(* IEC 61131-3 sources: sphere-usecases/water-treatment/implementations/openplc/projects/simulator_project, 4 files *)

(* ---- simulator_clean.st ---- *)
TYPE
  HMI_UDT : STRUCT
    Start_PB : BOOL;
    Stop_PB : BOOL;
    Start_Active : BOOL;
    Stop_Active : BOOL;
  END_STRUCT;
  P1_UDT : STRUCT
    RW_Tank_tnk_lvl : REAL;
    RW_Pump_flow : REAL;
    RW_Tank_PR_Valve_sts : BOOL;
    RW_Tank_P6B_Valve_sts : BOOL;
    RW_Tank_P_Valve_sts : BOOL;
    RW_Pump_sts : BOOL;
    RW_Pump_fault : BOOL;
    RW_Pump : REAL;
    RW_Tank_PR_Valve : BOOL;
    RW_Tank_P_Valve : BOOL;
    RW_Pump_start : BOOL;
    RW_Pump_stop : BOOL;
    RW_Tank_P6B_Valve : BOOL;
  END_STRUCT;
  P2_UDT : STRUCT
    ChemTreat_NaCl_Tank_tnk_lvl : REAL;
    ChemTreat_NaOCl_Tank_tnk_lvl : REAL;
    ChemTreat_HCl_Tank_tnk_lvl : REAL;
    ChemTreat_NaCl_Tank_Valve_sts : BOOL;
    ChemTreat_NaOCl_Tank_Valve_sts : BOOL;
    ChemTreat_HCl_Tank_Valve_sts : BOOL;
    ChemTreat_NaCl_Tank_Valve : BOOL;
    ChemTreat_NaOCl_Tank_Valve : BOOL;
    ChemTreat_HCl_Tank_Valve : BOOL;
  END_STRUCT;
  P3_UDT : STRUCT
    Ultrafiltration_UFFT_Tank_tnk_lvl : REAL;
    Ultrafiltration_UFFT_Tank_Valve_sts : BOOL;
    Ultrafiltration_UF_Drain_Valve_sts : BOOL;
    Ultrafiltration_UF_ROFT_Valve_sts : BOOL;
    Ultrafiltration_UF_BWP_Valve_sts : BOOL;
    Ultrafiltration_UFFT_Tank_Valve : BOOL;
    Ultrafiltration_UF_Drain_Valve : BOOL;
    Ultrafiltration_UF_ROFT_Valve : BOOL;
    Ultrafiltration_UF_BWP_Valve : BOOL;
  END_STRUCT;
  Phases_UDT : STRUCT
    Filling : BOOL;
    Draining : BOOL;
  END_STRUCT;
  RW_tank_AL_UDT : STRUCT
    LL_alarm : BOOL;
    L_alarm : BOOL;
    H_alarm : BOOL;
    HH_alarm : BOOL;
  END_STRUCT;
  System_State_UDT : STRUCT
    IDLE : BOOL;
    START : BOOL;
    RUNNING : BOOL;
    SHUTDOWN : BOOL;
    Permissives : ARRAY [0..31] OF BOOL;
    Permissives_Ready : BOOL;
  END_STRUCT;
  SYS_MESSAGES : STRUCT
    ProgramScanTime : DINT;
    AvailableMemory : REAL;
    ControllerStatus : SINT;
    ScanTime : REAL;
  END_STRUCT;
END_TYPE

PROGRAM MainProgram
  VAR_INPUT
    Alarms : RW_tank_AL_UDT;
    GSV_Message : SYS_MESSAGES;
    HMI : HMI_UDT;
    P1 : P1_UDT;
    P1_SYS : System_State_UDT;
    P2 : P2_UDT;
    P3 : P3_UDT;
  END_VAR
  VAR_INPUT
    di_2_0 AT %IX2.0 : BOOL;
    di_2_1 AT %IX2.1 : BOOL;
    di_2_10 AT %IX2.10 : BOOL;
    di_2_11 AT %IX2.11 : BOOL;
    di_2_2 AT %IX2.2 : BOOL;
    di_2_3 AT %IX2.3 : BOOL;
    di_2_4 AT %IX2.4 : BOOL;
    di_2_5 AT %IX2.5 : BOOL;
    di_2_6 AT %IX2.6 : BOOL;
    di_2_8 AT %IX2.8 : BOOL;
    di_2_9 AT %IX2.9 : BOOL;
    ai_7_0 AT %IW70 : REAL;
    di_7_ch0halarm AT %IX7.0 : BOOL;
    di_7_ch0hhalarm AT %IX7.0 : BOOL;
    di_7_ch0lalarm AT %IX7.0 : BOOL;
    di_7_ch0llalarm AT %IX7.0 : BOOL;
    ai_7_1 AT %IW71 : REAL;
    ai_7_2 AT %IW72 : REAL;
    ai_7_3 AT %IW73 : REAL;
    ai_7_4 AT %IW74 : REAL;
    ai_7_5 AT %IW75 : REAL;
  END_VAR
  VAR_OUTPUT
    ao_10_0 AT %QW100 : REAL;
    do_5_0 AT %QX5.0 : BOOL;
    do_5_1 AT %QX5.1 : BOOL;
    do_5_10 AT %QX5.10 : BOOL;
    do_5_11 AT %QX5.11 : BOOL;
    do_5_2 AT %QX5.2 : BOOL;
    do_5_3 AT %QX5.3 : BOOL;
    do_5_4 AT %QX5.4 : BOOL;
    do_5_5 AT %QX5.5 : BOOL;
    do_5_6 AT %QX5.6 : BOOL;
    do_5_7 AT %QX5.7 : BOOL;
    do_5_8 AT %QX5.8 : BOOL;
    do_5_9 AT %QX5.9 : BOOL;
  END_VAR

  (* IO_setup *)
  (* P1 Analog Input *)
  P1.RW_Tank_tnk_lvl := ai_7_0;
  P1.RW_Pump_flow := ai_7_1;
  (* P1 Digital Input *)
  P1.RW_Tank_PR_Valve_sts := di_2_0;
  P1.RW_Tank_P6B_Valve_sts := di_2_1;
  P1.RW_Tank_P_Valve_sts := di_2_2;
  P1.RW_Pump_sts := di_2_3;
  P1.RW_Pump_fault := di_2_4;
  (* P1 Analog Output *)
  P1.RW_Pump := ao_10_0;
  (* Digital Output *)
  P1.RW_Tank_PR_Valve := do_5_0;
  P1.RW_Tank_P6B_Valve := do_5_1;
  P1.RW_Tank_P_Valve := do_5_2;
  P1.RW_Pump_start := do_5_3;
  P1.RW_Pump_stop := do_5_4;
  (* P1 raw water tank alarms *)
  Alarms.LL_alarm := di_7_ch0llalarm;
  Alarms.L_alarm := di_7_ch0lalarm;
  Alarms.H_alarm := di_7_ch0halarm;
  Alarms.HH_alarm := di_7_ch0hhalarm;
  (* P2 Analog Input *)
  P2.ChemTreat_NaCl_Tank_tnk_lvl := ai_7_2;
  P2.ChemTreat_NaOCl_Tank_tnk_lvl := ai_7_3;
  P2.ChemTreat_HCl_Tank_tnk_lvl := ai_7_4;
  (* P2 Digital Input *)
  P2.ChemTreat_NaCl_Tank_Valve_sts := di_2_5;
  P2.ChemTreat_NaOCl_Tank_Valve_sts := di_2_6;
  (* P2 Analog Output *)
  (* NONE *)
  (* P2 Digital Output *)
  P2.ChemTreat_NaCl_Tank_Valve := do_5_5;
  P2.ChemTreat_NaOCl_Tank_Valve := do_5_6;
  P2.ChemTreat_HCl_Tank_Valve := do_5_7;
  (* P3 Analog Input *)
  P3.Ultrafiltration_UFFT_Tank_tnk_lvl := ai_7_5;
  (* P3 Digital Input *)
  P3.Ultrafiltration_UFFT_Tank_Valve_sts := di_2_8;
  P3.Ultrafiltration_UF_Drain_Valve_sts := di_2_9;
  P3.Ultrafiltration_UF_Drain_Valve_sts := di_2_10;
  P3.Ultrafiltration_UF_BWP_Valve_sts := di_2_11;
  (* P3 Analog Output *)
  (* none *)
  (* P3 Digital Output *)
  P3.Ultrafiltration_UFFT_Tank_Valve := do_5_8;
  P3.Ultrafiltration_UF_Drain_Valve := do_5_9;
  P3.Ultrafiltration_UF_ROFT_Valve := do_5_10;
  P3.Ultrafiltration_UF_BWP_Valve := do_5_11;

  (* Raw_water_control *)
  if P1.RW_Tank_tnk_lvl = 250.0 and P1_SYS.RUNNING then
  P1.RW_Pump_stop := True;
  P1.RW_Pump_start := False; (* send the outputs *)
  Alarms.LL_alarm := True;
  (* if the level is at 500 or lower than 500 open the valve *)
  elsif P1.RW_Tank_tnk_lvl <= 500.0 and P1_SYS.RUNNING then
  (* output to turn the valve open *)
  P1.RW_Tank_PR_Valve := True;
  Alarms.L_alarm := True;
  (* if level is at 800 *)
  elsif  P1.RW_Tank_tnk_lvl = 800.0 and P1_SYS.RUNNING then
  P1.RW_Tank_PR_Valve := False; (* close the valve *)
  Alarms.H_alarm := True;
  elsif P1.RW_Tank_tnk_lvl = 1200.0 and P1_SYS.RUNNING then
  Alarms.HH_alarm := True; (* if the tank is higher than or equal to 1200 set the high high alarm *)
  end_if;

  (* Raw_water_pump *)
  if P3.Ultrafiltration_UFFT_Tank_tnk_lvl = 800.0 AND P1_SYS.RUNNING then
  (* start the pump and open the valve from the other tank *)
  P1.RW_Tank_P_Valve := True;
  P1.RW_Pump_start := True;
  P1.RW_Pump_stop := False;
  elsif P3.Ultrafiltration_UFFT_Tank_tnk_lvl = 1000.0 AND P1_SYS.RUNNING then
  (* stop the pump and close the valve *)
  P1.RW_Tank_P_Valve := False;
  P1.RW_Pump_stop := True;
  P1.RW_Pump_start := False;
  end_if;

  (* State_change *)
  if not HMI.Start_Active AND not HMI.Stop_Active then
  (* if start and stop is not pressed go to idle *)
  P1_SYS.IDLE := True;
  P1_SYS.START := False;
  P1_SYS.RUNNING := False;
  P1_SYS.SHUTDOWN := False;
  elsif  HMI.Start_Active AND not HMI.Stop_Active then
  (* if the start pb and stop is not pressed then change the state of process one to starting *)
  P1_SYS.IDLE := False;
  P1_SYS.START := True;
  P1_SYS.RUNNING := False;
  P1_SYS.SHUTDOWN := False;
  (* if the tank level is greater than 250 at the start and UFFT is less than a 1000 we can start *)
  (* then and all permissves cond together into one tag so we know the plant is ready to start *)
  P1_SYS.Permissives_Ready := P1_SYS.Permissives[0] AND P1_SYS.Permissives[1];
  elsif HMI.Start_Active AND P1_SYS.Permissives_Ready then
  (* if the start was pressed and permissives are ready start running Process one *)
  P1_SYS.IDLE := False;
  P1_SYS.START := False;
  P1_SYS.RUNNING := True;
  P1_SYS.SHUTDOWN := False;
  elsif HMI.Stop_Active then
  (* if the stop button is pressed then go to shutdown state *)
  P1_SYS.IDLE := False;
  P1_SYS.START := False;
  P1_SYS.RUNNING := False;
  P1_SYS.SHUTDOWN := True;
  (* set all permissives to false *)
  P1_SYS.Permissives_Ready := False;
  end_if;
END_PROGRAM

CONFIGURATION config
  VAR_GLOBAL
    ao_10_0 AT %QW100 : REAL;
    di_2_0 AT %IX2.0 : BOOL;
    di_2_1 AT %IX2.1 : BOOL;
    di_2_10 AT %IX2.10 : BOOL;
    di_2_11 AT %IX2.11 : BOOL;
    di_2_2 AT %IX2.2 : BOOL;
    di_2_3 AT %IX2.3 : BOOL;
    di_2_4 AT %IX2.4 : BOOL;
    di_2_5 AT %IX2.5 : BOOL;
    di_2_6 AT %IX2.6 : BOOL;
    di_2_8 AT %IX2.8 : BOOL;
    di_2_9 AT %IX2.9 : BOOL;
    do_5_0 AT %QX5.0 : BOOL;
    do_5_1 AT %QX5.1 : BOOL;
    do_5_10 AT %QX5.10 : BOOL;
    do_5_11 AT %QX5.11 : BOOL;
    do_5_2 AT %QX5.2 : BOOL;
    do_5_3 AT %QX5.3 : BOOL;
    do_5_4 AT %QX5.4 : BOOL;
    do_5_5 AT %QX5.5 : BOOL;
    do_5_6 AT %QX5.6 : BOOL;
    do_5_7 AT %QX5.7 : BOOL;
    do_5_8 AT %QX5.8 : BOOL;
    do_5_9 AT %QX5.9 : BOOL;
    ai_7_0 AT %IW70 : REAL;
    di_7_ch0halarm AT %IX7.0 : BOOL;
    di_7_ch0hhalarm AT %IX7.0 : BOOL;
    di_7_ch0lalarm AT %IX7.0 : BOOL;
    di_7_ch0llalarm AT %IX7.0 : BOOL;
    ai_7_1 AT %IW71 : REAL;
    ai_7_2 AT %IW72 : REAL;
    ai_7_3 AT %IW73 : REAL;
    ai_7_4 AT %IW74 : REAL;
    ai_7_5 AT %IW75 : REAL;
  END_VAR

  RESOURCE res_MainProgram ON PLC
    TASK task_MainProgram(INTERVAL := T#100ms,PRIORITY := 0);
    PROGRAM MainProgram_instance : MainProgram;
  END_RESOURCE
END_CONFIGURATION

(* ---- simulator_final.st ---- *)
PROGRAM SimulatorProgram
  VAR
    (* ===== Internal physics state ===== *)
    rw_tank_level : REAL := 600.0;
    uf_tank_level : REAL := 400.0;
    nacl_level : REAL := 800.0;
    naocl_level : REAL := 800.0;
    hcl_level : REAL := 800.0;
    pump_running : BOOL := FALSE;
    pump_flow : REAL := 0.0;

    (* Valve status with delay timers *)
    pr_valve_open : BOOL := FALSE;
    pr_valve_timer : INT := 0;
    p6b_valve_open : BOOL := FALSE;
    p6b_valve_timer : INT := 0;
    p_valve_open : BOOL := FALSE;
    p_valve_timer : INT := 0;
    nacl_valve_open : BOOL := FALSE;
    nacl_valve_timer : INT := 0;
    naocl_valve_open : BOOL := FALSE;
    naocl_valve_timer : INT := 0;
    hcl_valve_open : BOOL := FALSE;
    hcl_valve_timer : INT := 0;
    uf_valve_open : BOOL := FALSE;
    uf_valve_timer : INT := 0;
    uf_drain_open : BOOL := FALSE;
    uf_drain_timer : INT := 0;
    uf_roft_open : BOOL := FALSE;
    uf_roft_timer : INT := 0;
    uf_bwp_open : BOOL := FALSE;
    uf_bwp_timer : INT := 0;

    init_done : BOOL := FALSE;
    pump_timer : INT := 0;
    pump_requested : BOOL := FALSE;
    admin_reset_seq_seen : INT := 0;
    admin_apply_seq_seen : INT := 0;

    (* ===== Constants ===== *)
    DT_SEC : REAL := 0.1;            (* 100ms scan interval *)
    PUMP_MAX_FLOW : REAL := 120.0;   (* L/min at 100% speed *)
    PR_INFLOW_RATE : REAL := 50.0;   (* L/min from external source *)
    DOSING_RATE : REAL := 5.0;       (* L/min chemical drain *)
    UF_DRAIN_RATE : REAL := 30.0;    (* L/min UF drain/ROFT *)
    VALVE_DELAY : INT := 5;          (* cycles = 500ms *)
    PUMP_DELAY : INT := 8;           (* cycles = 800ms *)
    RW_TANK_MAX : REAL := 1500.0;
    UF_TANK_MAX : REAL := 1200.0;
    CHEM_TANK_MAX : REAL := 1000.0;
  END_VAR
  VAR_EXTERNAL
    (* ===== Bridge command inputs - written by external bridge ===== *)
    cmd_pr_valve : INT;      (* 0/1  PR valve command *)
    cmd_p6b_valve : INT;     (* 0/1  P6B valve command *)
    cmd_p_valve : INT;       (* 0/1  Process valve command *)
    cmd_pump_start : INT;    (* 0/1  Pump start *)
    cmd_pump_stop : INT;     (* 0/1  Pump stop *)
    cmd_nacl_valve : INT;    (* 0/1  NaCl valve command *)
    cmd_naocl_valve : INT;   (* 0/1  NaOCl valve command *)
    cmd_hcl_valve : INT;     (* 0/1  HCl valve command *)
    cmd_uf_valve : INT;      (* 0/1  UF tank valve command *)
    cmd_uf_drain : INT;      (* 0/1  UF drain valve command *)
    cmd_uf_roft : INT;       (* 0/1  UF ROFT valve command *)
    cmd_uf_bwp : INT;        (* 0/1  UF BWP valve command *)
    cmd_pump_speed : INT;    (* 0-100  pump speed % *)
    admin_init_rw_level : INT;   (* reset baseline: RW tank level *)
    admin_init_uf_level : INT;   (* reset baseline: UF tank level *)
    admin_init_nacl_level : INT; (* reset baseline: NaCl tank *)
    admin_init_naocl_level : INT;(* reset baseline: NaOCl tank *)
    admin_init_hcl_level : INT;  (* reset baseline: HCl tank *)
    admin_reset_seq : INT;       (* increments trigger full sim reset *)
    admin_apply_rw_level : INT;  (* runtime RW level override *)
    admin_apply_uf_level : INT;  (* runtime UF level override *)
    admin_apply_nacl_level : INT;(* runtime NaCl level override *)
    admin_apply_naocl_level : INT;(* runtime NaOCl level override *)
    admin_apply_hcl_level : INT; (* runtime HCl level override *)
    admin_apply_rw_flag : INT;   (* 0/1 apply override *)
    admin_apply_uf_flag : INT;
    admin_apply_nacl_flag : INT;
    admin_apply_naocl_flag : INT;
    admin_apply_hcl_flag : INT;
    admin_apply_seq : INT;       (* increments trigger level apply *)

    (* ===== Bridge sensor outputs - read by bridge ===== *)
    out_rw_level : INT;      (* RW tank level mm *)
    out_rw_flow : INT;       (* RW pump flow L/min *)
    out_nacl_level : INT;    (* NaCl tank level mm *)
    out_naocl_level : INT;   (* NaOCl tank level mm *)
    out_hcl_level : INT;     (* HCl tank level mm *)
    out_uf_level : INT;      (* UF tank level mm *)
    out_pr_valve_sts : INT;  (* 0/1 *)
    out_p6b_valve_sts : INT;
    out_p_valve_sts : INT;
    out_pump_sts : INT;
    out_pump_fault : INT;
    out_nacl_valve_sts : INT;
    out_naocl_valve_sts : INT;
    out_hcl_valve_sts : INT;
    out_uf_valve_sts : INT;
    out_uf_drain_sts : INT;
    out_uf_roft_sts : INT;
    out_uf_bwp_sts : INT;
  END_VAR

  IF NOT init_done THEN
    rw_tank_level := 600.0;
    uf_tank_level := 400.0;
    nacl_level := 800.0;
    naocl_level := 800.0;
    hcl_level := 800.0;
    pump_running := FALSE;
    pump_flow := 0.0;
    pr_valve_open := FALSE;
    pr_valve_timer := 0;
    p6b_valve_open := FALSE;
    p6b_valve_timer := 0;
    p_valve_open := FALSE;
    p_valve_timer := 0;
    nacl_valve_open := FALSE;
    nacl_valve_timer := 0;
    naocl_valve_open := FALSE;
    naocl_valve_timer := 0;
    hcl_valve_open := FALSE;
    hcl_valve_timer := 0;
    uf_valve_open := FALSE;
    uf_valve_timer := 0;
    uf_drain_open := FALSE;
    uf_drain_timer := 0;
    uf_roft_open := FALSE;
    uf_roft_timer := 0;
    uf_bwp_open := FALSE;
    uf_bwp_timer := 0;
    pump_timer := 0;
    pump_requested := FALSE;
    admin_reset_seq_seen := admin_reset_seq;
    admin_apply_seq_seen := admin_apply_seq;
    init_done := TRUE;
  END_IF;

  (* ========================================================= *)
  (* 0. Testbed admin hooks                                    *)
  (*    These registers let the host reset or perturb the sim  *)
  (*    without rebuilding images or restarting the stack.     *)
  (* ========================================================= *)
  IF admin_reset_seq <> admin_reset_seq_seen THEN
    admin_reset_seq_seen := admin_reset_seq;
    rw_tank_level := INT_TO_REAL(admin_init_rw_level);
    uf_tank_level := INT_TO_REAL(admin_init_uf_level);
    nacl_level := INT_TO_REAL(admin_init_nacl_level);
    naocl_level := INT_TO_REAL(admin_init_naocl_level);
    hcl_level := INT_TO_REAL(admin_init_hcl_level);
    pump_running := FALSE;
    pump_flow := 0.0;
    pr_valve_open := FALSE;
    pr_valve_timer := 0;
    p6b_valve_open := FALSE;
    p6b_valve_timer := 0;
    p_valve_open := FALSE;
    p_valve_timer := 0;
    nacl_valve_open := FALSE;
    nacl_valve_timer := 0;
    naocl_valve_open := FALSE;
    naocl_valve_timer := 0;
    hcl_valve_open := FALSE;
    hcl_valve_timer := 0;
    uf_valve_open := FALSE;
    uf_valve_timer := 0;
    uf_drain_open := FALSE;
    uf_drain_timer := 0;
    uf_roft_open := FALSE;
    uf_roft_timer := 0;
    uf_bwp_open := FALSE;
    uf_bwp_timer := 0;
    pump_timer := 0;
    pump_requested := FALSE;
  END_IF;

  IF admin_apply_seq <> admin_apply_seq_seen THEN
    admin_apply_seq_seen := admin_apply_seq;
    IF admin_apply_rw_flag <> 0 THEN
      rw_tank_level := INT_TO_REAL(admin_apply_rw_level);
    END_IF;
    IF admin_apply_uf_flag <> 0 THEN
      uf_tank_level := INT_TO_REAL(admin_apply_uf_level);
    END_IF;
    IF admin_apply_nacl_flag <> 0 THEN
      nacl_level := INT_TO_REAL(admin_apply_nacl_level);
    END_IF;
    IF admin_apply_naocl_flag <> 0 THEN
      naocl_level := INT_TO_REAL(admin_apply_naocl_level);
    END_IF;
    IF admin_apply_hcl_flag <> 0 THEN
      hcl_level := INT_TO_REAL(admin_apply_hcl_level);
    END_IF;
  END_IF;

  (* ========================================================= *)
  (* 1. Update valve status with delay                         *)
  (* ========================================================= *)

  (* PR valve *)
  IF cmd_pr_valve <> 0 THEN
    IF NOT pr_valve_open THEN
      pr_valve_timer := pr_valve_timer + 1;
      IF pr_valve_timer >= VALVE_DELAY THEN
        pr_valve_open := TRUE;
        pr_valve_timer := 0;
      END_IF;
    END_IF;
  ELSE
    IF pr_valve_open THEN
      pr_valve_timer := pr_valve_timer + 1;
      IF pr_valve_timer >= VALVE_DELAY THEN
        pr_valve_open := FALSE;
        pr_valve_timer := 0;
      END_IF;
    ELSE
      pr_valve_timer := 0;
    END_IF;
  END_IF;

  (* P6B valve *)
  IF cmd_p6b_valve <> 0 THEN
    IF NOT p6b_valve_open THEN
      p6b_valve_timer := p6b_valve_timer + 1;
      IF p6b_valve_timer >= VALVE_DELAY THEN
        p6b_valve_open := TRUE;
        p6b_valve_timer := 0;
      END_IF;
    END_IF;
  ELSE
    IF p6b_valve_open THEN
      p6b_valve_timer := p6b_valve_timer + 1;
      IF p6b_valve_timer >= VALVE_DELAY THEN
        p6b_valve_open := FALSE;
        p6b_valve_timer := 0;
      END_IF;
    ELSE
      p6b_valve_timer := 0;
    END_IF;
  END_IF;

  (* P valve *)
  IF cmd_p_valve <> 0 THEN
    IF NOT p_valve_open THEN
      p_valve_timer := p_valve_timer + 1;
      IF p_valve_timer >= VALVE_DELAY THEN
        p_valve_open := TRUE;
        p_valve_timer := 0;
      END_IF;
    END_IF;
  ELSE
    IF p_valve_open THEN
      p_valve_timer := p_valve_timer + 1;
      IF p_valve_timer >= VALVE_DELAY THEN
        p_valve_open := FALSE;
        p_valve_timer := 0;
      END_IF;
    ELSE
      p_valve_timer := 0;
    END_IF;
  END_IF;

  (* NaCl valve *)
  IF cmd_nacl_valve <> 0 THEN
    IF NOT nacl_valve_open THEN
      nacl_valve_timer := nacl_valve_timer + 1;
      IF nacl_valve_timer >= VALVE_DELAY THEN
        nacl_valve_open := TRUE;
        nacl_valve_timer := 0;
      END_IF;
    END_IF;
  ELSE
    IF nacl_valve_open THEN
      nacl_valve_timer := nacl_valve_timer + 1;
      IF nacl_valve_timer >= VALVE_DELAY THEN
        nacl_valve_open := FALSE;
        nacl_valve_timer := 0;
      END_IF;
    ELSE
      nacl_valve_timer := 0;
    END_IF;
  END_IF;

  (* NaOCl valve *)
  IF cmd_naocl_valve <> 0 THEN
    IF NOT naocl_valve_open THEN
      naocl_valve_timer := naocl_valve_timer + 1;
      IF naocl_valve_timer >= VALVE_DELAY THEN
        naocl_valve_open := TRUE;
        naocl_valve_timer := 0;
      END_IF;
    END_IF;
  ELSE
    IF naocl_valve_open THEN
      naocl_valve_timer := naocl_valve_timer + 1;
      IF naocl_valve_timer >= VALVE_DELAY THEN
        naocl_valve_open := FALSE;
        naocl_valve_timer := 0;
      END_IF;
    ELSE
      naocl_valve_timer := 0;
    END_IF;
  END_IF;

  (* HCl valve *)
  IF cmd_hcl_valve <> 0 THEN
    IF NOT hcl_valve_open THEN
      hcl_valve_timer := hcl_valve_timer + 1;
      IF hcl_valve_timer >= VALVE_DELAY THEN
        hcl_valve_open := TRUE;
        hcl_valve_timer := 0;
      END_IF;
    END_IF;
  ELSE
    IF hcl_valve_open THEN
      hcl_valve_timer := hcl_valve_timer + 1;
      IF hcl_valve_timer >= VALVE_DELAY THEN
        hcl_valve_open := FALSE;
        hcl_valve_timer := 0;
      END_IF;
    ELSE
      hcl_valve_timer := 0;
    END_IF;
  END_IF;

  (* UF tank valve *)
  IF cmd_uf_valve <> 0 THEN
    IF NOT uf_valve_open THEN
      uf_valve_timer := uf_valve_timer + 1;
      IF uf_valve_timer >= VALVE_DELAY THEN
        uf_valve_open := TRUE;
        uf_valve_timer := 0;
      END_IF;
    END_IF;
  ELSE
    IF uf_valve_open THEN
      uf_valve_timer := uf_valve_timer + 1;
      IF uf_valve_timer >= VALVE_DELAY THEN
        uf_valve_open := FALSE;
        uf_valve_timer := 0;
      END_IF;
    ELSE
      uf_valve_timer := 0;
    END_IF;
  END_IF;

  (* UF drain valve *)
  IF cmd_uf_drain <> 0 THEN
    IF NOT uf_drain_open THEN
      uf_drain_timer := uf_drain_timer + 1;
      IF uf_drain_timer >= VALVE_DELAY THEN
        uf_drain_open := TRUE;
        uf_drain_timer := 0;
      END_IF;
    END_IF;
  ELSE
    IF uf_drain_open THEN
      uf_drain_timer := uf_drain_timer + 1;
      IF uf_drain_timer >= VALVE_DELAY THEN
        uf_drain_open := FALSE;
        uf_drain_timer := 0;
      END_IF;
    ELSE
      uf_drain_timer := 0;
    END_IF;
  END_IF;

  (* UF ROFT valve *)
  IF cmd_uf_roft <> 0 THEN
    IF NOT uf_roft_open THEN
      uf_roft_timer := uf_roft_timer + 1;
      IF uf_roft_timer >= VALVE_DELAY THEN
        uf_roft_open := TRUE;
        uf_roft_timer := 0;
      END_IF;
    END_IF;
  ELSE
    IF uf_roft_open THEN
      uf_roft_timer := uf_roft_timer + 1;
      IF uf_roft_timer >= VALVE_DELAY THEN
        uf_roft_open := FALSE;
        uf_roft_timer := 0;
      END_IF;
    ELSE
      uf_roft_timer := 0;
    END_IF;
  END_IF;

  (* UF BWP valve *)
  IF cmd_uf_bwp <> 0 THEN
    IF NOT uf_bwp_open THEN
      uf_bwp_timer := uf_bwp_timer + 1;
      IF uf_bwp_timer >= VALVE_DELAY THEN
        uf_bwp_open := TRUE;
        uf_bwp_timer := 0;
      END_IF;
    END_IF;
  ELSE
    IF uf_bwp_open THEN
      uf_bwp_timer := uf_bwp_timer + 1;
      IF uf_bwp_timer >= VALVE_DELAY THEN
        uf_bwp_open := FALSE;
        uf_bwp_timer := 0;
      END_IF;
    ELSE
      uf_bwp_timer := 0;
    END_IF;
  END_IF;

  (* ========================================================= *)
  (* 2. Update pump status with delay                          *)
  (* ========================================================= *)
  pump_requested := cmd_pump_start <> 0 AND cmd_pump_stop = 0;

  IF pump_requested AND NOT pump_running THEN
    pump_timer := pump_timer + 1;
    IF pump_timer >= PUMP_DELAY THEN
      pump_running := TRUE;
      pump_timer := 0;
    END_IF;
  ELSIF NOT pump_requested AND pump_running THEN
    pump_timer := pump_timer + 1;
    IF pump_timer >= PUMP_DELAY THEN
      pump_running := FALSE;
      pump_timer := 0;
    END_IF;
  ELSE
    pump_timer := 0;
  END_IF;

  (* ========================================================= *)
  (* 3. Compute flows                                          *)
  (* ========================================================= *)
  IF pump_running THEN
    pump_flow := INT_TO_REAL(cmd_pump_speed) * PUMP_MAX_FLOW / 100.0;
    IF pump_flow < 0.0 THEN
      pump_flow := 0.0;
    END_IF;
    IF pump_flow > PUMP_MAX_FLOW THEN
      pump_flow := PUMP_MAX_FLOW;
    END_IF;
  ELSE
    pump_flow := 0.0;
  END_IF;

  (* ========================================================= *)
  (* 4. Tank mass balance - P1: Raw Water                      *)
  (*    inflow: PR valve open -> external source               *)
  (*    outflow: pump + P valve -> UF tank                     *)
  (* ========================================================= *)
  IF pr_valve_open THEN
    rw_tank_level := rw_tank_level + PR_INFLOW_RATE * DT_SEC / 60.0;
  END_IF;
  IF pump_running AND p_valve_open THEN
    rw_tank_level := rw_tank_level - pump_flow * DT_SEC / 60.0;
  END_IF;
  IF rw_tank_level < 0.0 THEN
    rw_tank_level := 0.0;
  END_IF;
  IF rw_tank_level > RW_TANK_MAX THEN
    rw_tank_level := RW_TANK_MAX;
  END_IF;

  (* ========================================================= *)
  (* 5. Tank mass balance - P2: Chemical tanks                 *)
  (*    drain when valve open, no inflow modeled               *)
  (* ========================================================= *)
  IF nacl_valve_open THEN
    nacl_level := nacl_level - DOSING_RATE * DT_SEC / 60.0;
  END_IF;
  IF nacl_level < 0.0 THEN
    nacl_level := 0.0;
  END_IF;
  IF nacl_level > CHEM_TANK_MAX THEN
    nacl_level := CHEM_TANK_MAX;
  END_IF;

  IF naocl_valve_open THEN
    naocl_level := naocl_level - DOSING_RATE * DT_SEC / 60.0;
  END_IF;
  IF naocl_level < 0.0 THEN
    naocl_level := 0.0;
  END_IF;
  IF naocl_level > CHEM_TANK_MAX THEN
    naocl_level := CHEM_TANK_MAX;
  END_IF;

  IF hcl_valve_open THEN
    hcl_level := hcl_level - DOSING_RATE * DT_SEC / 60.0;
  END_IF;
  IF hcl_level < 0.0 THEN
    hcl_level := 0.0;
  END_IF;
  IF hcl_level > CHEM_TANK_MAX THEN
    hcl_level := CHEM_TANK_MAX;
  END_IF;

  (* ========================================================= *)
  (* 6. Tank mass balance - P3: UF tank                        *)
  (*    inflow from P1 pump when P valve open                  *)
  (*    outflow via drain and ROFT valves                      *)
  (* ========================================================= *)
  IF pump_running AND p_valve_open THEN
    uf_tank_level := uf_tank_level + pump_flow * DT_SEC / 60.0;
  END_IF;
  IF uf_drain_open THEN
    uf_tank_level := uf_tank_level - UF_DRAIN_RATE * DT_SEC / 60.0;
  END_IF;
  IF uf_roft_open THEN
    uf_tank_level := uf_tank_level - UF_DRAIN_RATE * DT_SEC / 60.0;
  END_IF;
  IF uf_tank_level < 0.0 THEN
    uf_tank_level := 0.0;
  END_IF;
  IF uf_tank_level > UF_TANK_MAX THEN
    uf_tank_level := UF_TANK_MAX;
  END_IF;

  (* ========================================================= *)
  (* 7. Write outputs to bridge registers                      *)
  (* ========================================================= *)
  out_rw_level := REAL_TO_INT(rw_tank_level);
  out_rw_flow := REAL_TO_INT(pump_flow);
  out_nacl_level := REAL_TO_INT(nacl_level);
  out_naocl_level := REAL_TO_INT(naocl_level);
  out_hcl_level := REAL_TO_INT(hcl_level);
  out_uf_level := REAL_TO_INT(uf_tank_level);

  IF pr_valve_open THEN
    out_pr_valve_sts := 1;
  ELSE
    out_pr_valve_sts := 0;
  END_IF;
  IF p6b_valve_open THEN
    out_p6b_valve_sts := 1;
  ELSE
    out_p6b_valve_sts := 0;
  END_IF;
  IF p_valve_open THEN
    out_p_valve_sts := 1;
  ELSE
    out_p_valve_sts := 0;
  END_IF;
  IF pump_running THEN
    out_pump_sts := 1;
  ELSE
    out_pump_sts := 0;
  END_IF;
  out_pump_fault := 0;  (* no fault model yet *)
  IF nacl_valve_open THEN
    out_nacl_valve_sts := 1;
  ELSE
    out_nacl_valve_sts := 0;
  END_IF;
  IF naocl_valve_open THEN
    out_naocl_valve_sts := 1;
  ELSE
    out_naocl_valve_sts := 0;
  END_IF;
  IF hcl_valve_open THEN
    out_hcl_valve_sts := 1;
  ELSE
    out_hcl_valve_sts := 0;
  END_IF;
  IF uf_valve_open THEN
    out_uf_valve_sts := 1;
  ELSE
    out_uf_valve_sts := 0;
  END_IF;
  IF uf_drain_open THEN
    out_uf_drain_sts := 1;
  ELSE
    out_uf_drain_sts := 0;
  END_IF;
  IF uf_roft_open THEN
    out_uf_roft_sts := 1;
  ELSE
    out_uf_roft_sts := 0;
  END_IF;
  IF uf_bwp_open THEN
    out_uf_bwp_sts := 1;
  ELSE
    out_uf_bwp_sts := 0;
  END_IF;

END_PROGRAM

CONFIGURATION Config0
  VAR_GLOBAL
    (* Bridge command inputs *)
    cmd_pr_valve AT %QW200 : INT;
    cmd_p6b_valve AT %QW201 : INT;
    cmd_p_valve AT %QW202 : INT;
    cmd_pump_start AT %QW203 : INT;
    cmd_pump_stop AT %QW204 : INT;
    cmd_nacl_valve AT %QW205 : INT;
    cmd_naocl_valve AT %QW206 : INT;
    cmd_hcl_valve AT %QW207 : INT;
    cmd_uf_valve AT %QW208 : INT;
    cmd_uf_drain AT %QW209 : INT;
    cmd_uf_roft AT %QW210 : INT;
    cmd_uf_bwp AT %QW211 : INT;
    cmd_pump_speed AT %QW220 : INT;
    admin_init_rw_level AT %QW340 : INT;
    admin_init_uf_level AT %QW341 : INT;
    admin_init_nacl_level AT %QW342 : INT;
    admin_init_naocl_level AT %QW343 : INT;
    admin_init_hcl_level AT %QW344 : INT;
    admin_reset_seq AT %QW349 : INT;
    admin_apply_rw_level AT %QW360 : INT;
    admin_apply_uf_level AT %QW361 : INT;
    admin_apply_nacl_level AT %QW362 : INT;
    admin_apply_naocl_level AT %QW363 : INT;
    admin_apply_hcl_level AT %QW364 : INT;
    admin_apply_rw_flag AT %QW365 : INT;
    admin_apply_uf_flag AT %QW366 : INT;
    admin_apply_nacl_flag AT %QW367 : INT;
    admin_apply_naocl_flag AT %QW368 : INT;
    admin_apply_hcl_flag AT %QW369 : INT;
    admin_apply_seq AT %QW370 : INT;
    (* Bridge sensor outputs *)
    out_rw_level AT %QW300 : INT;
    out_rw_flow AT %QW301 : INT;
    out_nacl_level AT %QW302 : INT;
    out_naocl_level AT %QW303 : INT;
    out_hcl_level AT %QW304 : INT;
    out_uf_level AT %QW305 : INT;
    out_pr_valve_sts AT %QW320 : INT;
    out_p6b_valve_sts AT %QW321 : INT;
    out_p_valve_sts AT %QW322 : INT;
    out_pump_sts AT %QW323 : INT;
    out_pump_fault AT %QW324 : INT;
    out_nacl_valve_sts AT %QW325 : INT;
    out_naocl_valve_sts AT %QW326 : INT;
    out_hcl_valve_sts AT %QW327 : INT;
    out_uf_valve_sts AT %QW328 : INT;
    out_uf_drain_sts AT %QW329 : INT;
    out_uf_roft_sts AT %QW330 : INT;
    out_uf_bwp_sts AT %QW331 : INT;
  END_VAR

  RESOURCE Res0 ON PLC
    TASK task_SimulatorProgram(INTERVAL := T#100ms, PRIORITY := 0);
    PROGRAM SimulatorProgram_instance : SimulatorProgram;
  END_RESOURCE
END_CONFIGURATION

(* ---- simulator_fixed.st ---- *)
TYPE
  HMI_UDT : STRUCT
    Start_PB : BOOL;
    Stop_PB : BOOL;
    Start_Active : BOOL;
    Stop_Active : BOOL;
  END_STRUCT;
  P1_UDT : STRUCT
    RW_Tank_tnk_lvl : REAL;
    RW_Pump_flow : REAL;
    RW_Tank_PR_Valve_sts : BOOL;
    RW_Tank_P6B_Valve_sts : BOOL;
    RW_Tank_P_Valve_sts : BOOL;
    RW_Pump_sts : BOOL;
    RW_Pump_fault : BOOL;
    RW_Pump : REAL;
    RW_Tank_PR_Valve : BOOL;
    RW_Tank_P_Valve : BOOL;
    RW_Pump_start : BOOL;
    RW_Pump_stop : BOOL;
    RW_Tank_P6B_Valve : BOOL;
  END_STRUCT;
  P2_UDT : STRUCT
    ChemTreat_NaCl_Tank_tnk_lvl : REAL;
    ChemTreat_NaOCl_Tank_tnk_lvl : REAL;
    ChemTreat_HCl_Tank_tnk_lvl : REAL;
    ChemTreat_NaCl_Tank_Valve_sts : BOOL;
    ChemTreat_NaOCl_Tank_Valve_sts : BOOL;
    ChemTreat_HCl_Tank_Valve_sts : BOOL;
    ChemTreat_NaCl_Tank_Valve : BOOL;
    ChemTreat_NaOCl_Tank_Valve : BOOL;
    ChemTreat_HCl_Tank_Valve : BOOL;
  END_STRUCT;
  P3_UDT : STRUCT
    Ultrafiltration_UFFT_Tank_tnk_lvl : REAL;
    Ultrafiltration_UFFT_Tank_Valve_sts : BOOL;
    Ultrafiltration_UF_Drain_Valve_sts : BOOL;
    Ultrafiltration_UF_ROFT_Valve_sts : BOOL;
    Ultrafiltration_UF_BWP_Valve_sts : BOOL;
    Ultrafiltration_UFFT_Tank_Valve : BOOL;
    Ultrafiltration_UF_Drain_Valve : BOOL;
    Ultrafiltration_UF_ROFT_Valve : BOOL;
    Ultrafiltration_UF_BWP_Valve : BOOL;
  END_STRUCT;
  Phases_UDT : STRUCT
    Filling : BOOL;
    Draining : BOOL;
  END_STRUCT;
  RW_tank_AL_UDT : STRUCT
    LL_alarm : BOOL;
    L_alarm : BOOL;
    H_alarm : BOOL;
    HH_alarm : BOOL;
  END_STRUCT;
  System_State_UDT : STRUCT
    IDLE : BOOL;
    START : BOOL;
    RUNNING : BOOL;
    SHUTDOWN : BOOL;
    Permissives : ARRAY [0..31] OF BOOL;
    Permissives_Ready : BOOL;
  END_STRUCT;
  SYS_MESSAGES : STRUCT
    ProgramScanTime : DINT;
    AvailableMemory : REAL;
    ControllerStatus : SINT;
    ScanTime : REAL;
  END_STRUCT;
END_TYPE

PROGRAM MainProgram
  VAR_INPUT
    Alarms : RW_tank_AL_UDT;
    GSV_Message : SYS_MESSAGES;
    HMI : HMI_UDT;
    P1 : P1_UDT;
    P1_SYS : System_State_UDT;
    P2 : P2_UDT;
    P3 : P3_UDT;
  END_VAR
  VAR_INPUT
    di_2_0 : BOOL;
    di_2_1 : BOOL;
    di_2_10 : BOOL;
    di_2_11 : BOOL;
    di_2_2 : BOOL;
    di_2_3 : BOOL;
    di_2_4 : BOOL;
    di_2_5 : BOOL;
    di_2_6 : BOOL;
    di_2_8 : BOOL;
    di_2_9 : BOOL;
    ai_7_0 : REAL;
    di_7_ch0halarm : BOOL;
    di_7_ch0hhalarm : BOOL;
    di_7_ch0lalarm : BOOL;
    di_7_ch0llalarm : BOOL;
    ai_7_1 : REAL;
    ai_7_2 : REAL;
    ai_7_3 : REAL;
    ai_7_4 : REAL;
    ai_7_5 : REAL;
  END_VAR
  VAR_OUTPUT
    ao_10_0 : REAL;
    do_5_0 : BOOL;
    do_5_1 : BOOL;
    do_5_10 : BOOL;
    do_5_11 : BOOL;
    do_5_2 : BOOL;
    do_5_3 : BOOL;
    do_5_4 : BOOL;
    do_5_5 : BOOL;
    do_5_6 : BOOL;
    do_5_7 : BOOL;
    do_5_8 : BOOL;
    do_5_9 : BOOL;
  END_VAR

  (* IO_setup *)
  (* P1 Analog Input *)
  P1.RW_Tank_tnk_lvl := ai_7_0;
  P1.RW_Pump_flow := ai_7_1;
  (* P1 Digital Input *)
  P1.RW_Tank_PR_Valve_sts := di_2_0;
  P1.RW_Tank_P6B_Valve_sts := di_2_1;
  P1.RW_Tank_P_Valve_sts := di_2_2;
  P1.RW_Pump_sts := di_2_3;
  P1.RW_Pump_fault := di_2_4;
  (* P1 Analog Output *)
  P1.RW_Pump := ao_10_0;
  (* Digital Output *)
  P1.RW_Tank_PR_Valve := do_5_0;
  P1.RW_Tank_P6B_Valve := do_5_1;
  P1.RW_Tank_P_Valve := do_5_2;
  P1.RW_Pump_start := do_5_3;
  P1.RW_Pump_stop := do_5_4;
  (* P1 raw water tank alarms *)
  Alarms.LL_alarm := di_7_ch0llalarm;
  Alarms.L_alarm := di_7_ch0lalarm;
  Alarms.H_alarm := di_7_ch0halarm;
  Alarms.HH_alarm := di_7_ch0hhalarm;
  (* P2 Analog Input *)
  P2.ChemTreat_NaCl_Tank_tnk_lvl := ai_7_2;
  P2.ChemTreat_NaOCl_Tank_tnk_lvl := ai_7_3;
  P2.ChemTreat_HCl_Tank_tnk_lvl := ai_7_4;
  (* P2 Digital Input *)
  P2.ChemTreat_NaCl_Tank_Valve_sts := di_2_5;
  P2.ChemTreat_NaOCl_Tank_Valve_sts := di_2_6;
  (* P2 Analog Output *)
  (* NONE *)
  (* P2 Digital Output *)
  P2.ChemTreat_NaCl_Tank_Valve := do_5_5;
  P2.ChemTreat_NaOCl_Tank_Valve := do_5_6;
  P2.ChemTreat_HCl_Tank_Valve := do_5_7;
  (* P3 Analog Input *)
  P3.Ultrafiltration_UFFT_Tank_tnk_lvl := ai_7_5;
  (* P3 Digital Input *)
  P3.Ultrafiltration_UFFT_Tank_Valve_sts := di_2_8;
  P3.Ultrafiltration_UF_Drain_Valve_sts := di_2_9;
  P3.Ultrafiltration_UF_Drain_Valve_sts := di_2_10;
  P3.Ultrafiltration_UF_BWP_Valve_sts := di_2_11;
  (* P3 Analog Output *)
  (* none *)
  (* P3 Digital Output *)
  P3.Ultrafiltration_UFFT_Tank_Valve := do_5_8;
  P3.Ultrafiltration_UF_Drain_Valve := do_5_9;
  P3.Ultrafiltration_UF_ROFT_Valve := do_5_10;
  P3.Ultrafiltration_UF_BWP_Valve := do_5_11;

  (* Raw_water_control *)
  if P1.RW_Tank_tnk_lvl = 250.0 and P1_SYS.RUNNING then
  P1.RW_Pump_stop := True;
  P1.RW_Pump_start := False; (* send the outputs *)
  Alarms.LL_alarm := True;
  (* if the level is at 500 or lower than 500 open the valve *)
  elsif P1.RW_Tank_tnk_lvl <= 500.0 and P1_SYS.RUNNING then
  (* output to turn the valve open *)
  P1.RW_Tank_PR_Valve := True;
  Alarms.L_alarm := True;
  (* if level is at 800 *)
  elsif  P1.RW_Tank_tnk_lvl = 800.0 and P1_SYS.RUNNING then
  P1.RW_Tank_PR_Valve := False; (* close the valve *)
  Alarms.H_alarm := True;
  elsif P1.RW_Tank_tnk_lvl = 1200.0 and P1_SYS.RUNNING then
  Alarms.HH_alarm := True; (* if the tank is higher than or equal to 1200 set the high high alarm *)
  end_if;

  (* Raw_water_pump *)
  if P3.Ultrafiltration_UFFT_Tank_tnk_lvl = 800.0 AND P1_SYS.RUNNING then
  (* start the pump and open the valve from the other tank *)
  P1.RW_Tank_P_Valve := True;
  P1.RW_Pump_start := True;
  P1.RW_Pump_stop := False;
  elsif P3.Ultrafiltration_UFFT_Tank_tnk_lvl = 1000.0 AND P1_SYS.RUNNING then
  (* stop the pump and close the valve *)
  P1.RW_Tank_P_Valve := False;
  P1.RW_Pump_stop := True;
  P1.RW_Pump_start := False;
  end_if;

  (* State_change *)
  if not HMI.Start_Active AND not HMI.Stop_Active then
  (* if start and stop is not pressed go to idle *)
  P1_SYS.IDLE := True;
  P1_SYS.START := False;
  P1_SYS.RUNNING := False;
  P1_SYS.SHUTDOWN := False;
  elsif  HMI.Start_Active AND not HMI.Stop_Active then
  (* if the start pb and stop is not pressed then change the state of process one to starting *)
  P1_SYS.IDLE := False;
  P1_SYS.START := True;
  P1_SYS.RUNNING := False;
  P1_SYS.SHUTDOWN := False;
  (* if the tank level is greater than 250 at the start and UFFT is less than a 1000 we can start *)
  (* then and all permissves cond together into one tag so we know the plant is ready to start *)
  P1_SYS.Permissives_Ready := P1_SYS.Permissives[0] AND P1_SYS.Permissives[1];
  elsif HMI.Start_Active AND P1_SYS.Permissives_Ready then
  (* if the start was pressed and permissives are ready start running Process one *)
  P1_SYS.IDLE := False;
  P1_SYS.START := False;
  P1_SYS.RUNNING := True;
  P1_SYS.SHUTDOWN := False;
  elsif HMI.Stop_Active then
  (* if the stop button is pressed then go to shutdown state *)
  P1_SYS.IDLE := False;
  P1_SYS.START := False;
  P1_SYS.RUNNING := False;
  P1_SYS.SHUTDOWN := True;
  (* set all permissives to false *)
  P1_SYS.Permissives_Ready := False;
  end_if;
END_PROGRAM

CONFIGURATION config
  VAR_GLOBAL
    ao_10_0 : REAL;
    di_2_0 : BOOL;
    di_2_1 : BOOL;
    di_2_10 : BOOL;
    di_2_11 : BOOL;
    di_2_2 : BOOL;
    di_2_3 : BOOL;
    di_2_4 : BOOL;
    di_2_5 : BOOL;
    di_2_6 : BOOL;
    di_2_8 : BOOL;
    di_2_9 : BOOL;
    do_5_0 : BOOL;
    do_5_1 : BOOL;
    do_5_10 : BOOL;
    do_5_11 : BOOL;
    do_5_2 : BOOL;
    do_5_3 : BOOL;
    do_5_4 : BOOL;
    do_5_5 : BOOL;
    do_5_6 : BOOL;
    do_5_7 : BOOL;
    do_5_8 : BOOL;
    do_5_9 : BOOL;
    ai_7_0 : REAL;
    di_7_ch0halarm : BOOL;
    di_7_ch0hhalarm : BOOL;
    di_7_ch0lalarm : BOOL;
    di_7_ch0llalarm : BOOL;
    ai_7_1 : REAL;
    ai_7_2 : REAL;
    ai_7_3 : REAL;
    ai_7_4 : REAL;
    ai_7_5 : REAL;
  END_VAR

  RESOURCE res_MainProgram ON PLC
    TASK task_MainProgram(INTERVAL := T#100ms,PRIORITY := 0);
    PROGRAM MainProgram_instance : MainProgram;
  END_RESOURCE
END_CONFIGURATION

(* ---- simulator_st_file_to_upload.st ---- *)
TYPE
  HMI_UDT : STRUCT
    Start_PB : BOOL;
    Stop_PB : BOOL;
    Start_Active : BOOL;
    Stop_Active : BOOL;
  END_STRUCT;
  P1_UDT : STRUCT
    RW_Tank_tnk_lvl : REAL;
    RW_Pump_flow : REAL;
    RW_Tank_PR_Valve_sts : BOOL;
    RW_Tank_P6B_Valve_sts : BOOL;
    RW_Tank_P_Valve_sts : BOOL;
    RW_Pump_sts : BOOL;
    RW_Pump_fault : BOOL;
    RW_Pump : REAL;
    RW_Tank_PR_Valve : BOOL;
    RW_Tank_P_Valve : BOOL;
    RW_Pump_start : BOOL;
    RW_Pump_stop : BOOL;
    RW_Tank_P6B_Valve : BOOL;
  END_STRUCT;
  P2_UDT : STRUCT
    ChemTreat_NaCl_Tank_tnk_lvl : REAL;
    ChemTreat_NaOCl_Tank_tnk_lvl : REAL;
    ChemTreat_HCl_Tank_tnk_lvl : REAL;
    ChemTreat_NaCl_Tank_Valve_sts : BOOL;
    ChemTreat_NaOCl_Tank_Valve_sts : BOOL;
    ChemTreat_HCl_Tank_Valve_sts : BOOL;
    ChemTreat_NaCl_Tank_Valve : BOOL;
    ChemTreat_NaOCl_Tank_Valve : BOOL;
    ChemTreat_HCl_Tank_Valve : BOOL;
  END_STRUCT;
  P3_UDT : STRUCT
    Ultrafiltration_UFFT_Tank_tnk_lvl : REAL;
    Ultrafiltration_UFFT_Tank_Valve_sts : BOOL;
    Ultrafiltration_UF_Drain_Valve_sts : BOOL;
    Ultrafiltration_UF_ROFT_Valve_sts : BOOL;
    Ultrafiltration_UF_BWP_Valve_sts : BOOL;
    Ultrafiltration_UFFT_Tank_Valve : BOOL;
    Ultrafiltration_UF_Drain_Valve : BOOL;
    Ultrafiltration_UF_ROFT_Valve : BOOL;
    Ultrafiltration_UF_BWP_Valve : BOOL;
  END_STRUCT;
  Phases_UDT : STRUCT
    Filling : BOOL;
    Draining : BOOL;
  END_STRUCT;
  RW_tank_AL_UDT : STRUCT
    LL_alarm : BOOL;
    L_alarm : BOOL;
    H_alarm : BOOL;
    HH_alarm : BOOL;
  END_STRUCT;
  System_State_UDT : STRUCT
    IDLE : BOOL;
    START : BOOL;
    RUNNING : BOOL;
    SHUTDOWN : BOOL;
    Permissives : ARRAY [0..31] OF BOOL;
    Permissives_Ready : BOOL;
  END_STRUCT;
  SYS_MESSAGES : STRUCT
    ProgramScanTime : DINT;
    AvailableMemory : REAL;
    ControllerStatus : SINT;
    ScanTime : REAL;
  END_STRUCT;
END_TYPE

PROGRAM MainProgram
  VAR_INPUT
    Alarms : RW_tank_AL_UDT;
    GSV_Message : SYS_MESSAGES;
    HMI : HMI_UDT;
    P1 : P1_UDT;
    P1_SYS : System_State_UDT;
    P2 : P2_UDT;
    P3 : P3_UDT;
  END_VAR
  VAR_INPUT
    di_2_0 AT %IX2.0 : BOOL;
    di_2_1 AT %IX2.1 : BOOL;
    di_2_10 AT %IX2.10 : BOOL;
    di_2_11 AT %IX2.11 : BOOL;
    di_2_2 AT %IX2.2 : BOOL;
    di_2_3 AT %IX2.3 : BOOL;
    di_2_4 AT %IX2.4 : BOOL;
    di_2_5 AT %IX2.5 : BOOL;
    di_2_6 AT %IX2.6 : BOOL;
    di_2_8 AT %IX2.8 : BOOL;
    di_2_9 AT %IX2.9 : BOOL;
    ai_7_0 AT %IW70 : REAL;
    di_7_ch0halarm AT %IX7.0 : BOOL;
    di_7_ch0hhalarm AT %IX7.0 : BOOL;
    di_7_ch0lalarm AT %IX7.0 : BOOL;
    di_7_ch0llalarm AT %IX7.0 : BOOL;
    ai_7_1 AT %IW71 : REAL;
    ai_7_2 AT %IW72 : REAL;
    ai_7_3 AT %IW73 : REAL;
    ai_7_4 AT %IW74 : REAL;
    ai_7_5 AT %IW75 : REAL;
  END_VAR
  VAR_OUTPUT
    ao_10_0 AT %QW100 : REAL;
    do_5_0 AT %QX5.0 : BOOL;
    do_5_1 AT %QX5.1 : BOOL;
    do_5_10 AT %QX5.10 : BOOL;
    do_5_11 AT %QX5.11 : BOOL;
    do_5_2 AT %QX5.2 : BOOL;
    do_5_3 AT %QX5.3 : BOOL;
    do_5_4 AT %QX5.4 : BOOL;
    do_5_5 AT %QX5.5 : BOOL;
    do_5_6 AT %QX5.6 : BOOL;
    do_5_7 AT %QX5.7 : BOOL;
    do_5_8 AT %QX5.8 : BOOL;
    do_5_9 AT %QX5.9 : BOOL;
  END_VAR

  (* IO_setup *)
  (* P1 Analog Input *)
  P1.RW_Tank_tnk_lvl := ai_7_0;
  P1.RW_Pump_flow := ai_7_1;
  (* P1 Digital Input *)
  P1.RW_Tank_PR_Valve_sts := di_2_0;
  P1.RW_Tank_P6B_Valve_sts := di_2_1;
  P1.RW_Tank_P_Valve_sts := di_2_2;
  P1.RW_Pump_sts := di_2_3;
  P1.RW_Pump_fault := di_2_4;
  (* P1 Analog Output *)
  P1.RW_Pump := ao_10_0;
  (* Digital Output *)
  P1.RW_Tank_PR_Valve := do_5_0;
  P1.RW_Tank_P6B_Valve := do_5_1;
  P1.RW_Tank_P_Valve := do_5_2;
  P1.RW_Pump_start := do_5_3;
  P1.RW_Pump_stop := do_5_4;
  (* P1 raw water tank alarms *)
  Alarms.LL_alarm := di_7_ch0llalarm;
  Alarms.L_alarm := di_7_ch0lalarm;
  Alarms.H_alarm := di_7_ch0halarm;
  Alarms.HH_alarm := di_7_ch0hhalarm;
  (* P2 Analog Input *)
  P2.ChemTreat_NaCl_Tank_tnk_lvl := ai_7_2;
  P2.ChemTreat_NaOCl_Tank_tnk_lvl := ai_7_3;
  P2.ChemTreat_HCl_Tank_tnk_lvl := ai_7_4;
  (* P2 Digital Input *)
  P2.ChemTreat_NaCl_Tank_Valve_sts := di_2_5;
  P2.ChemTreat_NaOCl_Tank_Valve_sts := di_2_6;
  (* P2 Analog Output *)
  (* NONE *)
  (* P2 Digital Output *)
  P2.ChemTreat_NaCl_Tank_Valve := do_5_5;
  P2.ChemTreat_NaOCl_Tank_Valve := do_5_6;
  P2.ChemTreat_HCl_Tank_Valve := do_5_7;
  (* P3 Analog Input *)
  P3.Ultrafiltration_UFFT_Tank_tnk_lvl := ai_7_5;
  (* P3 Digital Input *)
  P3.Ultrafiltration_UFFT_Tank_Valve_sts := di_2_8;
  P3.Ultrafiltration_UF_Drain_Valve_sts := di_2_9;
  P3.Ultrafiltration_UF_Drain_Valve_sts := di_2_10;
  P3.Ultrafiltration_UF_BWP_Valve_sts := di_2_11;
  (* P3 Analog Output *)
  (* none *)
  (* P3 Digital Output *)
  P3.Ultrafiltration_UFFT_Tank_Valve := do_5_8;
  P3.Ultrafiltration_UF_Drain_Valve := do_5_9;
  P3.Ultrafiltration_UF_ROFT_Valve := do_5_10;
  P3.Ultrafiltration_UF_BWP_Valve := do_5_11;

  (* Raw_water_control *)
  if P1.RW_Tank_tnk_lvl = 250.0 and P1_SYS.RUNNING then
  P1.RW_Pump_stop := True;
  P1.RW_Pump_start := False; (* send the outputs *)
  Alarms.LL_alarm := True;
  (* if the level is at 500 or lower than 500 open the valve *)
  elsif P1.RW_Tank_tnk_lvl <= 500.0 and P1_SYS.RUNNING then
  (* output to turn the valve open *)
  P1.RW_Tank_PR_Valve := True;
  Alarms.L_alarm := True;
  (* if level is at 800 *)
  elsif  P1.RW_Tank_tnk_lvl = 800.0 and P1_SYS.RUNNING then
  P1.RW_Tank_PR_Valve := False; (* close the valve *)
  Alarms.H_alarm := True;
  elsif P1.RW_Tank_tnk_lvl = 1200.0 and P1_SYS.RUNNING then
  Alarms.HH_alarm := True; (* if the tank is higher than or equal to 1200 set the high high alarm *)
  end_if;

  (* Raw_water_pump *)
  if P3.Ultrafiltration_UFFT_Tank_tnk_lvl = 800.0 AND P1_SYS.RUNNING then
  (* start the pump and open the valve from the other tank *)
  P1.RW_Tank_P_Valve := True;
  P1.RW_Pump_start := True;
  P1.RW_Pump_stop := False;
  elsif P3.Ultrafiltration_UFFT_Tank_tnk_lvl = 1000.0 AND P1_SYS.RUNNING then
  (* stop the pump and close the valve *)
  P1.RW_Tank_P_Valve := False;
  P1.RW_Pump_stop := True;
  P1.RW_Pump_start := False;
  end_if;

  (* State_change *)
  if not HMI.Start_Active AND not HMI.Stop_Active then
  (* if start and stop is not pressed go to idle *)
  P1_SYS.IDLE := True;
  P1_SYS.START := False;
  P1_SYS.RUNNING := False;
  P1_SYS.SHUTDOWN := False;
  elsif  HMI.Start_Active AND not HMI.Stop_Active then
  (* if the start pb and stop is not pressed then change the state of process one to starting *)
  P1_SYS.IDLE := False;
  P1_SYS.START := True;
  P1_SYS.RUNNING := False;
  P1_SYS.SHUTDOWN := False;
  (* if the tank level is greater than 250 at the start and UFFT is less than a 1000 we can start *)
  (* then and all permissves cond together into one tag so we know the plant is ready to start *)
  P1_SYS.Permissives_Ready := P1_SYS.Permissives[0] AND P1_SYS.Permissives[1];
  elsif HMI.Start_Active AND P1_SYS.Permissives_Ready then
  (* if the start was pressed and permissives are ready start running Process one *)
  P1_SYS.IDLE := False;
  P1_SYS.START := False;
  P1_SYS.RUNNING := True;
  P1_SYS.SHUTDOWN := False;
  elsif HMI.Stop_Active then
  (* if the stop button is pressed then go to shutdown state *)
  P1_SYS.IDLE := False;
  P1_SYS.START := False;
  P1_SYS.RUNNING := False;
  P1_SYS.SHUTDOWN := True;
  (* set all permissives to false *)
  P1_SYS.Permissives_Ready := False;
  end_if;
END_PROGRAM

CONFIGURATION config
  VAR_GLOBAL
    ao_10_0 AT %QW100 : REAL;
    di_2_0 AT %IX2.0 : BOOL;
    di_2_1 AT %IX2.1 : BOOL;
    di_2_10 AT %IX2.10 : BOOL;
    di_2_11 AT %IX2.11 : BOOL;
    di_2_2 AT %IX2.2 : BOOL;
    di_2_3 AT %IX2.3 : BOOL;
    di_2_4 AT %IX2.4 : BOOL;
    di_2_5 AT %IX2.5 : BOOL;
    di_2_6 AT %IX2.6 : BOOL;
    di_2_8 AT %IX2.8 : BOOL;
    di_2_9 AT %IX2.9 : BOOL;
    do_5_0 AT %QX5.0 : BOOL;
    do_5_1 AT %QX5.1 : BOOL;
    do_5_10 AT %QX5.10 : BOOL;
    do_5_11 AT %QX5.11 : BOOL;
    do_5_2 AT %QX5.2 : BOOL;
    do_5_3 AT %QX5.3 : BOOL;
    do_5_4 AT %QX5.4 : BOOL;
    do_5_5 AT %QX5.5 : BOOL;
    do_5_6 AT %QX5.6 : BOOL;
    do_5_7 AT %QX5.7 : BOOL;
    do_5_8 AT %QX5.8 : BOOL;
    do_5_9 AT %QX5.9 : BOOL;
    ai_7_0 AT %IW70 : REAL;
    di_7_ch0halarm AT %IX7.0 : BOOL;
    di_7_ch0hhalarm AT %IX7.0 : BOOL;
    di_7_ch0lalarm AT %IX7.0 : BOOL;
    di_7_ch0llalarm AT %IX7.0 : BOOL;
    ai_7_1 AT %IW71 : REAL;
    ai_7_2 AT %IW72 : REAL;
    ai_7_3 AT %IW73 : REAL;
    ai_7_4 AT %IW74 : REAL;
    ai_7_5 AT %IW75 : REAL;
  END_VAR

  RESOURCE res_MainProgram ON PLC
    TASK task_MainProgram(INTERVAL := T#100ms,PRIORITY := 0);
    PROGRAM MainProgram_instance : MainProgram;
  END_RESOURCE
END_CONFIGURATION

(*DBG:char md5[] = "527971c67af0de80c69f5223004ec189";*)
(*DBG:/**)
(*DBG: * This file is part of OpenPLC Runtime*)
(*DBG: **)
(*DBG: * Copyright (C) 2023 Autonomy, GP Orcullo*)
(*DBG: * Based on the work by GP Orcullo on Beremiz for uC*)
(*DBG: **)
(*DBG: * This program is free software; you can redistribute it and/or*)
(*DBG: * modify it under the terms of the GNU General Public License*)
(*DBG: * as published by the Free Software Foundation; either version 2*)
(*DBG: * of the License, or (at your option) any later version.*)
(*DBG: **)
(*DBG: * This program is distributed in the hope that it will be useful,*)
(*DBG: * but WITHOUT ANY WARRANTY; without even the implied warranty of*)
(*DBG: * MERCHANTABILITY or FITNESS FOR A PARTICULAR PURPOSE.  See the*)
(*DBG: * GNU General Public License for more details.*)
(*DBG: **)
(*DBG: * You should have received a copy of the GNU General Public License*)
(*DBG: * along with this program; If not, see <http://www.gnu.org/licenses/>.*)
(*DBG: **)
(*DBG: */*)
(*DBG:*)
(*DBG:#include <stdbool.h>*)
(*DBG:*)
(*DBG:#include "iec_types_all.h"*)
(*DBG:#include "POUS.h"*)
(*DBG:*)
(*DBG:#define SAME_ENDIANNESS      0*)
(*DBG:#define REVERSE_ENDIANNESS   1*)
(*DBG:*)
(*DBG:uint8_t endianness;*)
(*DBG:*)
(*DBG:*)
(*DBG:extern __IEC_REAL_t CONFIG__AO_10_0;*)
(*DBG:extern __IEC_BOOL_t CONFIG__DI_2_0;*)
(*DBG:extern __IEC_BOOL_t CONFIG__DI_2_1;*)
(*DBG:extern __IEC_BOOL_t CONFIG__DI_2_10;*)
(*DBG:extern __IEC_BOOL_t CONFIG__DI_2_11;*)
(*DBG:extern __IEC_BOOL_t CONFIG__DI_2_2;*)
(*DBG:extern __IEC_BOOL_t CONFIG__DI_2_3;*)
(*DBG:extern __IEC_BOOL_t CONFIG__DI_2_4;*)
(*DBG:extern __IEC_BOOL_t CONFIG__DI_2_5;*)
(*DBG:extern __IEC_BOOL_t CONFIG__DI_2_6;*)
(*DBG:extern __IEC_BOOL_t CONFIG__DI_2_8;*)
(*DBG:extern __IEC_BOOL_t CONFIG__DI_2_9;*)
(*DBG:extern __IEC_BOOL_t CONFIG__DO_5_0;*)
(*DBG:extern __IEC_BOOL_t CONFIG__DO_5_1;*)
(*DBG:extern __IEC_BOOL_t CONFIG__DO_5_10;*)
(*DBG:extern __IEC_BOOL_t CONFIG__DO_5_11;*)
(*DBG:extern __IEC_BOOL_t CONFIG__DO_5_2;*)
(*DBG:extern __IEC_BOOL_t CONFIG__DO_5_3;*)
(*DBG:extern __IEC_BOOL_t CONFIG__DO_5_4;*)
(*DBG:extern __IEC_BOOL_t CONFIG__DO_5_5;*)
(*DBG:extern __IEC_BOOL_t CONFIG__DO_5_6;*)
(*DBG:extern __IEC_BOOL_t CONFIG__DO_5_7;*)
(*DBG:extern __IEC_BOOL_t CONFIG__DO_5_8;*)
(*DBG:extern __IEC_BOOL_t CONFIG__DO_5_9;*)
(*DBG:extern __IEC_REAL_t CONFIG__AI_7_0;*)
(*DBG:extern __IEC_BOOL_t CONFIG__DI_7_CH0HALARM;*)
(*DBG:extern __IEC_BOOL_t CONFIG__DI_7_CH0HHALARM;*)
(*DBG:extern __IEC_BOOL_t CONFIG__DI_7_CH0LALARM;*)
(*DBG:extern __IEC_BOOL_t CONFIG__DI_7_CH0LLALARM;*)
(*DBG:extern __IEC_REAL_t CONFIG__AI_7_1;*)
(*DBG:extern __IEC_REAL_t CONFIG__AI_7_2;*)
(*DBG:extern __IEC_REAL_t CONFIG__AI_7_3;*)
(*DBG:extern __IEC_REAL_t CONFIG__AI_7_4;*)
(*DBG:extern __IEC_REAL_t CONFIG__AI_7_5;*)
(*DBG:extern MAINPROGRAM RES_MAINPROGRAM__MAINPROGRAM_INSTANCE;*)
(*DBG:*)
(*DBG:static const struct {*)
(*DBG:    void *ptr;*)
(*DBG:    __IEC_types_enum type;*)
(*DBG:} debug_vars[] = {*)
(*DBG:    {&(CONFIG__AO_10_0), REAL_ENUM},*)
(*DBG:    {&(CONFIG__DI_2_0), BOOL_ENUM},*)
(*DBG:    {&(CONFIG__DI_2_1), BOOL_ENUM},*)
(*DBG:    {&(CONFIG__DI_2_10), BOOL_ENUM},*)
(*DBG:    {&(CONFIG__DI_2_11), BOOL_ENUM},*)
(*DBG:    {&(CONFIG__DI_2_2), BOOL_ENUM},*)
(*DBG:    {&(CONFIG__DI_2_3), BOOL_ENUM},*)
(*DBG:    {&(CONFIG__DI_2_4), BOOL_ENUM},*)
(*DBG:    {&(CONFIG__DI_2_5), BOOL_ENUM},*)
(*DBG:    {&(CONFIG__DI_2_6), BOOL_ENUM},*)
(*DBG:    {&(CONFIG__DI_2_8), BOOL_ENUM},*)
(*DBG:    {&(CONFIG__DI_2_9), BOOL_ENUM},*)
(*DBG:    {&(CONFIG__DO_5_0), BOOL_ENUM},*)
(*DBG:    {&(CONFIG__DO_5_1), BOOL_ENUM},*)
(*DBG:    {&(CONFIG__DO_5_10), BOOL_ENUM},*)
(*DBG:    {&(CONFIG__DO_5_11), BOOL_ENUM},*)
(*DBG:    {&(CONFIG__DO_5_2), BOOL_ENUM},*)
(*DBG:    {&(CONFIG__DO_5_3), BOOL_ENUM},*)
(*DBG:    {&(CONFIG__DO_5_4), BOOL_ENUM},*)
(*DBG:    {&(CONFIG__DO_5_5), BOOL_ENUM},*)
(*DBG:    {&(CONFIG__DO_5_6), BOOL_ENUM},*)
(*DBG:    {&(CONFIG__DO_5_7), BOOL_ENUM},*)
(*DBG:    {&(CONFIG__DO_5_8), BOOL_ENUM},*)
(*DBG:    {&(CONFIG__DO_5_9), BOOL_ENUM},*)
(*DBG:    {&(CONFIG__AI_7_0), REAL_ENUM},*)
(*DBG:    {&(CONFIG__DI_7_CH0HALARM), BOOL_ENUM},*)
(*DBG:    {&(CONFIG__DI_7_CH0HHALARM), BOOL_ENUM},*)
(*DBG:    {&(CONFIG__DI_7_CH0LALARM), BOOL_ENUM},*)
(*DBG:    {&(CONFIG__DI_7_CH0LLALARM), BOOL_ENUM},*)
(*DBG:    {&(CONFIG__AI_7_1), REAL_ENUM},*)
(*DBG:    {&(CONFIG__AI_7_2), REAL_ENUM},*)
(*DBG:    {&(CONFIG__AI_7_3), REAL_ENUM},*)
(*DBG:    {&(CONFIG__AI_7_4), REAL_ENUM},*)
(*DBG:    {&(CONFIG__AI_7_5), REAL_ENUM},*)
(*DBG:    {&(RES_MAINPROGRAM__MAINPROGRAM_INSTANCE.DI_2_0), BOOL_ENUM},*)
(*DBG:    {&(RES_MAINPROGRAM__MAINPROGRAM_INSTANCE.DI_2_1), BOOL_ENUM},*)
(*DBG:    {&(RES_MAINPROGRAM__MAINPROGRAM_INSTANCE.DI_2_10), BOOL_ENUM},*)
(*DBG:    {&(RES_MAINPROGRAM__MAINPROGRAM_INSTANCE.DI_2_11), BOOL_ENUM},*)
(*DBG:    {&(RES_MAINPROGRAM__MAINPROGRAM_INSTANCE.DI_2_2), BOOL_ENUM},*)
(*DBG:    {&(RES_MAINPROGRAM__MAINPROGRAM_INSTANCE.DI_2_3), BOOL_ENUM},*)
(*DBG:    {&(RES_MAINPROGRAM__MAINPROGRAM_INSTANCE.DI_2_4), BOOL_ENUM},*)
(*DBG:    {&(RES_MAINPROGRAM__MAINPROGRAM_INSTANCE.DI_2_5), BOOL_ENUM},*)
(*DBG:    {&(RES_MAINPROGRAM__MAINPROGRAM_INSTANCE.DI_2_6), BOOL_ENUM},*)
(*DBG:    {&(RES_MAINPROGRAM__MAINPROGRAM_INSTANCE.DI_2_8), BOOL_ENUM},*)
(*DBG:    {&(RES_MAINPROGRAM__MAINPROGRAM_INSTANCE.DI_2_9), BOOL_ENUM},*)
(*DBG:    {&(RES_MAINPROGRAM__MAINPROGRAM_INSTANCE.AI_7_0), REAL_ENUM},*)
(*DBG:    {&(RES_MAINPROGRAM__MAINPROGRAM_INSTANCE.DI_7_CH0HALARM), BOOL_ENUM},*)
(*DBG:    {&(RES_MAINPROGRAM__MAINPROGRAM_INSTANCE.DI_7_CH0HHALARM), BOOL_ENUM},*)
(*DBG:    {&(RES_MAINPROGRAM__MAINPROGRAM_INSTANCE.DI_7_CH0LALARM), BOOL_ENUM},*)
(*DBG:    {&(RES_MAINPROGRAM__MAINPROGRAM_INSTANCE.DI_7_CH0LLALARM), BOOL_ENUM},*)
(*DBG:    {&(RES_MAINPROGRAM__MAINPROGRAM_INSTANCE.AI_7_1), REAL_ENUM},*)
(*DBG:    {&(RES_MAINPROGRAM__MAINPROGRAM_INSTANCE.AI_7_2), REAL_ENUM},*)
(*DBG:    {&(RES_MAINPROGRAM__MAINPROGRAM_INSTANCE.AI_7_3), REAL_ENUM},*)
(*DBG:    {&(RES_MAINPROGRAM__MAINPROGRAM_INSTANCE.AI_7_4), REAL_ENUM},*)
(*DBG:    {&(RES_MAINPROGRAM__MAINPROGRAM_INSTANCE.AI_7_5), REAL_ENUM},*)
(*DBG:    {&(RES_MAINPROGRAM__MAINPROGRAM_INSTANCE.AO_10_0), REAL_ENUM},*)
(*DBG:    {&(RES_MAINPROGRAM__MAINPROGRAM_INSTANCE.DO_5_0), BOOL_ENUM},*)
(*DBG:    {&(RES_MAINPROGRAM__MAINPROGRAM_INSTANCE.DO_5_1), BOOL_ENUM},*)
(*DBG:    {&(RES_MAINPROGRAM__MAINPROGRAM_INSTANCE.DO_5_10), BOOL_ENUM},*)
(*DBG:    {&(RES_MAINPROGRAM__MAINPROGRAM_INSTANCE.DO_5_11), BOOL_ENUM},*)
(*DBG:    {&(RES_MAINPROGRAM__MAINPROGRAM_INSTANCE.DO_5_2), BOOL_ENUM},*)
(*DBG:    {&(RES_MAINPROGRAM__MAINPROGRAM_INSTANCE.DO_5_3), BOOL_ENUM},*)
(*DBG:    {&(RES_MAINPROGRAM__MAINPROGRAM_INSTANCE.DO_5_4), BOOL_ENUM},*)
(*DBG:    {&(RES_MAINPROGRAM__MAINPROGRAM_INSTANCE.DO_5_5), BOOL_ENUM},*)
(*DBG:    {&(RES_MAINPROGRAM__MAINPROGRAM_INSTANCE.DO_5_6), BOOL_ENUM},*)
(*DBG:    {&(RES_MAINPROGRAM__MAINPROGRAM_INSTANCE.DO_5_7), BOOL_ENUM},*)
(*DBG:    {&(RES_MAINPROGRAM__MAINPROGRAM_INSTANCE.DO_5_8), BOOL_ENUM},*)
(*DBG:    {&(RES_MAINPROGRAM__MAINPROGRAM_INSTANCE.DO_5_9), BOOL_ENUM},*)
(*DBG:};*)
(*DBG:*)
(*DBG:#define VAR_COUNT               68*)
(*DBG:*)
(*DBG:uint16_t get_var_count(void)*)
(*DBG:{*)
(*DBG:    return VAR_COUNT;*)
(*DBG:}*)
(*DBG:*)
(*DBG:size_t get_var_size(size_t idx)*)
(*DBG:{*)
(*DBG:    if (idx >= VAR_COUNT)*)
(*DBG:    {*)
(*DBG:        return 0;*)
(*DBG:    }*)
(*DBG:    switch (debug_vars[idx].type) {*)
(*DBG:    case REAL_ENUM:*)
(*DBG:        return sizeof(REAL);*)
(*DBG:    case BOOL_ENUM:*)
(*DBG:        return sizeof(BOOL);*)
(*DBG:    default:*)
(*DBG:        return 0;*)
(*DBG:    }*)
(*DBG:}*)
(*DBG:*)
(*DBG:void *get_var_addr(size_t idx)*)
(*DBG:{*)
(*DBG:    void *ptr = debug_vars[idx].ptr;*)
(*DBG:*)
(*DBG:    switch (debug_vars[idx].type) {*)
(*DBG:    case REAL_ENUM:*)
(*DBG:        return (void *)&((__IEC_REAL_t *) ptr)->value;*)
(*DBG:    case BOOL_ENUM:*)
(*DBG:        return (void *)&((__IEC_BOOL_t *) ptr)->value;*)
(*DBG:    default:*)
(*DBG:        return 0;*)
(*DBG:    }*)
(*DBG:}*)
(*DBG:*)
(*DBG:void force_var(size_t idx, bool forced, void *val)*)
(*DBG:{*)
(*DBG:    void *ptr = debug_vars[idx].ptr;*)
(*DBG:*)
(*DBG:    if (forced) {*)
(*DBG:        size_t var_size = get_var_size(idx);*)
(*DBG:        switch (debug_vars[idx].type) {*)
(*DBG:        case REAL_ENUM: {*)
(*DBG:            memcpy(&((__IEC_REAL_t *) ptr)->value, val, var_size);*)
(*DBG:            //((__IEC_REAL_t *) ptr)->value = *((REAL *) val);*)
(*DBG:            ((__IEC_REAL_t *) ptr)->flags |= __IEC_FORCE_FLAG;*)
(*DBG:            break;*)
(*DBG:        }*)
(*DBG:        case BOOL_ENUM: {*)
(*DBG:            memcpy(&((__IEC_BOOL_t *) ptr)->value, val, var_size);*)
(*DBG:            //((__IEC_BOOL_t *) ptr)->value = *((BOOL *) val);*)
(*DBG:            ((__IEC_BOOL_t *) ptr)->flags |= __IEC_FORCE_FLAG;*)
(*DBG:            break;*)
(*DBG:        }*)
(*DBG:        default:*)
(*DBG:            break;*)
(*DBG:        }*)
(*DBG:    } else {*)
(*DBG:        switch (debug_vars[idx].type) {*)
(*DBG:        case REAL_ENUM:*)
(*DBG:            ((__IEC_REAL_t *) ptr)->flags &= ~__IEC_FORCE_FLAG;*)
(*DBG:            break;*)
(*DBG:        case BOOL_ENUM:*)
(*DBG:            ((__IEC_BOOL_t *) ptr)->flags &= ~__IEC_FORCE_FLAG;*)
(*DBG:            break;*)
(*DBG:        default:*)
(*DBG:            break;*)
(*DBG:        }*)
(*DBG:    }*)
(*DBG:}*)
(*DBG:*)
(*DBG:void swap_bytes(void *ptr, size_t size) *)
(*DBG:{*)
(*DBG:    uint8_t *bytePtr = (uint8_t *)ptr;*)
(*DBG:    size_t i;*)
(*DBG:    for (i = 0; i < size / 2; ++i) *)
(*DBG:    {*)
(*DBG:        uint8_t temp = bytePtr[i];*)
(*DBG:        bytePtr[i] = bytePtr[size - 1 - i];*)
(*DBG:        bytePtr[size - 1 - i] = temp;*)
(*DBG:    }*)
(*DBG:}*)
(*DBG:*)
(*DBG:void trace_reset(void)*)
(*DBG:{*)
(*DBG:    for (size_t i=0; i < VAR_COUNT; i++) *)
(*DBG:    {*)
(*DBG:        force_var(i, false, 0);*)
(*DBG:    }*)
(*DBG:}*)
(*DBG:*)
(*DBG:void set_trace(size_t idx, bool forced, void *val)*)
(*DBG:{*)
(*DBG:    if (idx >= 0 && idx < VAR_COUNT) *)
(*DBG:    {*)
(*DBG:        if (endianness == REVERSE_ENDIANNESS)*)
(*DBG:        {*)
(*DBG:            // Aaaaarghhhh... Stupid AVR is Big Endian.*)
(*DBG:            swap_bytes(val, get_var_size(idx));*)
(*DBG:        }*)
(*DBG:*)
(*DBG:        force_var(idx, forced, val);*)
(*DBG:    }*)
(*DBG:}*)
(*DBG:*)
(*DBG:void set_endianness(uint8_t value)*)
(*DBG:{*)
(*DBG:    if (value == SAME_ENDIANNESS || value == REVERSE_ENDIANNESS)*)
(*DBG:    {*)
(*DBG:        endianness = value;*)
(*DBG:    }*)
(*DBG:}*)
(*DBG:*)
